///////////////////////////////////////////////////////////////////////////////
// function calls                                                            //
///////////////////////////////////////////////////////////////////////////////
      CALL "ALARM_SQ" (
// <- meta.block.fc.body meta.block.network
// ^^^^^^^^^^^^^^^^^^^^ meta.block.fc.body meta.block.network
//    ^^^^ meta.function-call - meta.function-call meta.function-call
//        ^^^^^^^^^^^^ meta.function-call.name - meta.function-call meta.function-call
//                    ^ meta.function-call.arguments - meta.function-call meta.function-call
//    ^^^^ keyword.control.call
//         ^ meta.string.s7.awl string.quoted.double.s7.awl punctuation.definition.string.begin.s7.awl - variable
//          ^^^^^^^^ meta.string.s7.awl variable.function.symbol.s7.awl - string
//                  ^ meta.string.s7.awl string.quoted.double.s7.awl punctuation.definition.string.end.s7.awl - variable
//                    ^ punctuation.section.parens.begin
           EN      := L 4.0,
// <- meta.block.fc.body meta.block.network meta.function-call.arguments
// ^^^^^^^^^^^^^^^^^^^^^^^^^^ meta.block.fc.body meta.block.network meta.function-call.arguments
//         ^^^^^^^^  meta.mapping.key
//                 ^^ meta.mapping - meta.mapping.key - meta.mapping.value
//                   ^^^^^ meta.mapping.value - meta.mapping.key
//                        ^ meta.mapping
//         ^^ variable.parameter
//                 ^^ punctuation.separator.key-value
//                    ^^^^^ variable.language.address.s7.awl
//                         ^ punctuation.separator.mapping.pair.s7.awl
           INTF    := DB 2,
// <- meta.block.fc.body meta.block.network meta.function-call.arguments
// ^^^^^^^^^^^^^^^^^^^^^^^^^^ meta.block.fc.body meta.block.network meta.function-call.arguments
//         ^^^^^^^^  meta.mapping.key
//                 ^^ meta.mapping - meta.mapping.key - meta.mapping.value
//                   ^^^^^ meta.mapping.value - meta.mapping.key
//                        ^ meta.mapping
//         ^^^^ variable.parameter
//                 ^^ punctuation.separator.key-value
//                    ^^^^ variable.language.db.s7.awl
           TMR     := T 2,
// <- meta.block.fc.body meta.block.network meta.function-call.arguments
// ^^^^^^^^^^^^^^^^^^^^^^^^^^ meta.block.fc.body meta.block.network meta.function-call.arguments
//         ^^^^^^^^  meta.mapping.key
//                 ^^ meta.mapping - meta.mapping.key - meta.mapping.value
//                   ^^^^ meta.mapping.value - meta.mapping.key
//                       ^ meta.mapping
//         ^^^ variable.parameter
//                 ^^ punctuation.separator.key-value
//                    ^^^ variable.language.timer.s7.awl
           CNT     := Z 2,
// <- meta.block.fc.body meta.block.network meta.function-call.arguments
// ^^^^^^^^^^^^^^^^^^^^^^^^^^ meta.block.fc.body meta.block.network meta.function-call.arguments
//         ^^^^^^^^  meta.mapping.key
//                 ^^ meta.mapping - meta.mapping.key - meta.mapping.value
//                   ^^^^ meta.mapping.value - meta.mapping.key
//                       ^ meta.mapping
//         ^^^ variable.parameter
//                 ^^ punctuation.separator.key-value
//                    ^^^ variable.language.counter.s7.awl
           SIG     := "msgs".A700127,
// <- meta.block.fc.body meta.block.network meta.function-call.arguments
// ^^^^^^^^^^^^^^^^^^^^^^^^^^^^^^^^^^ meta.block.fc.body meta.block.network meta.function-call.arguments
//         ^^^^^^^^  meta.mapping.key
//                 ^^ meta.mapping - meta.mapping.key - meta.mapping.value
//                   ^^^^^^^^^^^^^^^ meta.mapping.value - meta.mapping.key
//                                  ^ meta.mapping
//         ^^^ variable.parameter
//                 ^^ punctuation.separator.key-value
//                    ^ string.quoted.double punctuation.definition.string.begin - variable
//                    ^^^^^^ meta.string
//                     ^^^^ variable.other.symbol - string
//                         ^ string.quoted.double punctuation.definition.string.end - variable
//                          ^ punctuation.accessor
//                           ^^^^^^^ variable.other.member
//                                  ^ punctuation.separator.mapping.pair
           ID      := W#16#EEEE,
// <- meta.block.fc.body meta.block.network meta.function-call.arguments
// ^^^^^^^^^^^^^^^^^^^^^^^^^^^^^ meta.block.fc.body meta.block.network meta.function-call.arguments
//         ^^^^^^^^  meta.mapping.key
//                 ^^ meta.mapping - meta.mapping.key - meta.mapping.value
//                   ^^^^^^^^^^ meta.mapping.value - meta.mapping.key
//                             ^ meta.mapping
//         ^^ variable.parameter
//                 ^^ punctuation.separator.key-value
//                    ^^^^^^^^^ constant.numeric.integer.hexadecimal
//                             ^ punctuation.separator.mapping.pair
           EV_ID   := DW#16#AAEDF,
// <- meta.block.fc.body meta.block.network meta.function-call.arguments
// ^^^^^^^^^^^^^^^^^^^^^^^^^^^^^^ meta.block.fc.body meta.block.network meta.function-call.arguments
//         ^^^^^^^^  meta.mapping.key
//                 ^^ meta.mapping - meta.mapping.key - meta.mapping.value
//                   ^^^^^^^^^^^^ meta.mapping.value - meta.mapping.key
//                               ^ meta.mapping
//         ^^^^^ variable.parameter
//                 ^^ punctuation.separator.key-value
//                    ^^^^^^^^^^^ constant.numeric.integer.hexadecimal
//                               ^ punctuation.separator.mapping.pair
           ANY     := P# DB20.DBX40.0 WORD 10,
// <- meta.block.fc.body meta.block.network meta.function-call.arguments
// ^^^^^^^^^^^^^^^^^^^^^^^^^ meta.block.fc.body meta.block.network meta.function-call.arguments
//         ^^^^^^^^  meta.mapping.key
//                 ^^ meta.mapping - meta.mapping.key - meta.mapping.value
//                   ^^^^^^^^^^^^^^^^^^^^^^^^ meta.mapping.value - meta.mapping.key
//                                    ^^^^ storage.type.s7.awl
//                                           ^ meta.mapping
//         ^^ variable.parameter
//                 ^^ punctuation.separator.key-value
//                    ^^^^^^^^^^^^^^^^^^^^^^^ constant.language.any-pointer
           SD      := #data,
// <- meta.block.fc.body meta.block.network meta.function-call.arguments
// ^^^^^^^^^^^^^^^^^^^^^^^^^ meta.block.fc.body meta.block.network meta.function-call.arguments
//         ^^^^^^^^  meta.mapping.key
//                 ^^ meta.mapping - meta.mapping.key - meta.mapping.value
//                   ^^^^^^ meta.mapping.value - meta.mapping.key
//                         ^ meta.mapping
//         ^^ variable.parameter
//                 ^^ punctuation.separator.key-value
//                    ^ punctuation.definition.variable.begin
//                     ^^^^ variable.other.local
//                         ^ punctuation.separator.mapping.pair
           RET_VAL := MW200);
// <- meta.block.fc.body meta.block.network meta.function-call.arguments
// ^^^^^^^^^^^^^^^^^^^^^^^^^ meta.block.fc.body meta.block.network meta.function-call.arguments
//         ^^^^^^^^  meta.mapping.key
//                 ^^ meta.mapping - meta.mapping.key - meta.mapping.value
//                   ^^^^^^ meta.mapping.value - meta.mapping.key
//         ^^^^^^^ variable.parameter
//                 ^^ punctuation.separator.key-value
//                    ^^^^^ variable.language.address
//                         ^ punctuation.section.parens.end
//                          ^ punctuation.terminator.statement

   CALL FC 10 ();
// ^^^^ meta.function-call.s7.awl
//     ^^^^^^^ meta.function-call.name.s7.awl
//            ^^ meta.function-call.arguments.s7.awl
// ^^^^ keyword.control.call.s7.awl
//      ^^^^^ variable.function.address.s7.awl
//            ^ punctuation.section.parens.begin.s7.awl
//             ^ punctuation.section.parens.end.s7.awl

   CALL SFC 10 ();
// ^^^^ meta.function-call.s7.awl
//     ^^^^^^^^ meta.function-call.name.s7.awl
//             ^^ meta.function-call.arguments.s7.awl
// ^^^^ keyword.control.call.s7.awl
//      ^^^^^^ variable.function.address.s7.awl
//             ^ punctuation.section.parens.begin.s7.awl
//              ^ punctuation.section.parens.end.s7.awl

   CALL FB 10, DB 10 ();
// ^^^^ meta.function-call.s7.awl - meta.function-call meta.function-call
//     ^^^^^^^ meta.function-call.name.s7.awl - meta.function-call meta.function-call
//            ^^^^^^^ meta.function-call.instance.s7.awl - meta.function-call meta.function-call
//                   ^^ meta.function-call.arguments.s7.awl - meta.function-call meta.function-call
// ^^^^ keyword.control.call.s7.awl
//      ^^^^^ variable.function.address.s7.awl
//           ^ punctuation.separator.sequence.s7.awl
//             ^^^^^ variable.language.db.s7.awl
//                   ^ punctuation.section.parens.begin.s7.awl
//                    ^ punctuation.section.parens.end.s7.awl

   CALL "Block", "InstDB" ();
// ^^^^ meta.function-call.s7.awl - meta.function-call meta.function-call
//     ^^^^^^^^^ meta.function-call.name.s7.awl - meta.function-call meta.function-call
//              ^^^^^^^^^^ meta.function-call.instance.s7.awl - meta.function-call meta.function-call
//                        ^^ meta.function-call.arguments.s7.awl - meta.function-call meta.function-call
// ^^^^ keyword.control.call.s7.awl
//      ^ meta.string.s7.awl string.quoted.double.s7.awl punctuation.definition.string.begin.s7.awl - variable
//       ^^^^^ meta.string.s7.awl variable.function.symbol.s7.awl - string
//            ^ meta.string.s7.awl string.quoted.double.s7.awl punctuation.definition.string.end.s7.awl - variable
//             ^ punctuation.separator.sequence.s7.awl
//                ^^^^^^ variable.other.symbol.s7.awl
//                        ^ punctuation.section.parens.begin.s7.awl
//                         ^ punctuation.section.parens.end.s7.awl

   END_FUNCTION
// ^^^^^^^^^^^^ meta.block.fc.body
// ^^^^^^^^^^^^ keyword.other.fc.end
